(* IEC 61131-3 sources: PortalRobot/Portal_robot/Device/application/FB/FB_MULTI_TYPE, 3 files *)

(* ---- FB_MULTI_TYPE_CONFIG_MANAGER.st ---- *)
FUNCTION_BLOCK FB_MULTI_TYPE_CONFIG_MANAGER
VAR_INPUT
	xTestInitialize  : BOOL; // Атомарная загрузка конфигурации из тестового буфера
	stTestScenario   : ST_TEST_SCENARIO_BUFFER;
	Command          : ST_MULTI_TYPE_COMMAND; // Запросы конфигурации от HMI
	xCellRunning     : BOOL; // Автоматический цикл выполняется
	xMotionBusy      : BOOL; // Оси ещё движутся
	stRobotStatus    : ST_ROBOT_STATUS; // Состояние робота
	astMagazineStatus : ARRAY [1..GVL_CELL_SETTINGS.MagazineCount] OF ST_MAGAZINE_STATUS; // Оба магазина
	astMachineStatus : ARRAY [1..3] OF ST_MACHINE_PUBLIC; // Состояния станков
	uiRows           : UINT; // Строки активной матрицы
	uiColumns        : UINT; // Столбцы активной матрицы
END_VAR
VAR_OUTPUT
	Config : ST_MULTI_TYPE_CONFIG; // Фактически принятая конфигурация
	Status : ST_MULTI_TYPE_CONFIG_STATUS; // Разрешения и диагностика
END_VAR
VAR
	xInitialized        : BOOL; // Начальные безопасные значения заданы
	xAllMachinesSafe    : BOOL; // Станки не обслуживаются и не обрабатывают
	xAllMachinesDisabled: BOOL; // Все станки выключены
	xAllMagazinesEditable : BOOL; // Оба магазина выключены и не заняты
	xAllTypesHaveMachines : BOOL; // Каждый тип назначен хотя бы одному станку
	uiMachine           : UINT; // Индекс станка
	uiMagazine          : UINT; // Индекс магазина
	uiSlot              : UINT; // Индекс слота
	uiType              : UINT; // Индекс типа
	auiMachineCount     : ARRAY [1..3] OF UINT; // Количество станков каждого типа
	auiSlotCount        : ARRAY [1..3] OF UINT; // Количество слотов каждого типа
	rtSetTypeCount      : R_TRIG; // Фронт изменения количества типов
	rtSetMachineType    : R_TRIG; // Фронт назначения типа станку
	rtSetSlotType       : R_TRIG; // Фронт назначения типа слоту
	rtAutoDistribute    : R_TRIG; // Фронт автоматического распределения
END_VAR
VAR CONSTANT
	FIRST_MACHINE : UINT := UINT#1;
	LAST_MACHINE  : UINT := UINT#3;
	FIRST_TYPE    : UINT := UINT#1;
	LAST_TYPE     : UINT := UINT#3;
	WRN_TYPE_COUNT_NOT_ALLOWED : UINT := UINT#23;
	WRN_MACHINE_TYPE_REJECTED  : UINT := UINT#24;
	WRN_SLOT_TYPE_REJECTED     : UINT := UINT#25;
	WRN_DISTRIBUTION_REJECTED  : UINT := UINT#26;
END_VAR

// --- BEGIN IMPLEMENTATION ---

IF (uiRows > UINT#0)
AND (uiColumns > UINT#0)
AND ((uiRows * uiColumns) <= SINT_TO_UINT(GVL_CELL_SETTINGS.NumberDetail)) THEN
	Status.uiActiveSlotCount := uiRows * uiColumns;
ELSE
	Status.uiActiveSlotCount := UINT#0;
END_IF;

IF NOT xInitialized THEN
	Config.uiTypeCount := UINT#1;
	FOR uiMachine := FIRST_MACHINE TO LAST_MACHINE DO
		Config.auiMachineType[uiMachine] := UINT#1;
	END_FOR;
	FOR uiSlot := UINT#1 TO SINT_TO_UINT(GVL_CELL_SETTINGS.NumberDetail) DO
		IF uiSlot <= Status.uiActiveSlotCount THEN
			Config.auiSlotType[uiSlot] := UINT#1;
		ELSE
			Config.auiSlotType[uiSlot] := UINT#0;
		END_IF;
	END_FOR;
	xInitialized := TRUE;
END_IF;

xAllMachinesSafe := TRUE;
xAllMachinesDisabled := TRUE;
FOR uiMachine := FIRST_MACHINE TO LAST_MACHINE DO
	IF astMachineStatus[uiMachine].xBusy
	OR astMachineStatus[uiMachine].xProcessing THEN
		xAllMachinesSafe := FALSE;
	END_IF;
	IF astMachineStatus[uiMachine].xEnabled
	OR astMachineStatus[uiMachine].xDisablePending THEN
		xAllMachinesDisabled := FALSE;
	END_IF;
END_FOR;

xAllMagazinesEditable := TRUE;
FOR uiMagazine := UINT#1 TO INT_TO_UINT(GVL_CELL_SETTINGS.MagazineCount) DO
	IF astMagazineStatus[uiMagazine].xEnabled
	OR astMagazineStatus[uiMagazine].xBusy
	OR astMagazineStatus[uiMagazine].xDisablePending THEN
		xAllMagazinesEditable := FALSE;
	END_IF;
END_FOR;

Status.xMagazineConfigAllowed := NOT xCellRunning
	AND NOT xMotionBusy
	AND NOT stRobotStatus.xBusy
	AND NOT stRobotStatus.xBlankAvailable
	AND NOT stRobotStatus.xDetailAvailable
	AND xAllMagazinesEditable
	AND xAllMachinesSafe;
Status.xTypeCountAllowed := Status.xMagazineConfigAllowed
	AND xAllMachinesDisabled;

FOR uiMachine := FIRST_MACHINE TO LAST_MACHINE DO
	Status.axMachineTypeAllowed[uiMachine] := NOT xCellRunning
		AND NOT xMotionBusy
		AND NOT stRobotStatus.xBusy
		AND NOT stRobotStatus.xBlankAvailable
		AND NOT stRobotStatus.xDetailAvailable
		AND xAllMagazinesEditable
		AND NOT astMachineStatus[uiMachine].xEnabled
		AND NOT astMachineStatus[uiMachine].xDisablePending
		AND NOT astMachineStatus[uiMachine].xBusy
		AND NOT astMachineStatus[uiMachine].xProcessing;
END_FOR;

rtSetTypeCount(CLK := Command.xSetTypeCount);
rtSetMachineType(CLK := Command.xSetMachineType);
rtSetSlotType(CLK := Command.xSetSlotType);
rtAutoDistribute(CLK := Command.xAutoDistribute);

IF rtSetTypeCount.Q THEN
	IF NOT Status.xTypeCountAllowed
	OR (Command.uiRequestedTypeCount < FIRST_TYPE)
	OR (Command.uiRequestedTypeCount > LAST_TYPE) THEN
		RaiseWarning(uiCode := WRN_TYPE_COUNT_NOT_ALLOWED);
	ELSE
		Config.uiTypeCount := Command.uiRequestedTypeCount;
		CASE Config.uiTypeCount OF
			UINT#1:
				Config.auiMachineType[1] := UINT#1;
				Config.auiMachineType[2] := UINT#1;
				Config.auiMachineType[3] := UINT#1;
			UINT#2:
				Config.auiMachineType[1] := UINT#1;
				Config.auiMachineType[2] := UINT#1;
				Config.auiMachineType[3] := UINT#2;
			UINT#3:
				Config.auiMachineType[1] := UINT#1;
				Config.auiMachineType[2] := UINT#2;
				Config.auiMachineType[3] := UINT#3;
		END_CASE;
		ApplyDistribution();
	END_IF;
END_IF;

IF rtSetMachineType.Q THEN
	IF (Command.uiRequestedMachine < FIRST_MACHINE)
	OR (Command.uiRequestedMachine > LAST_MACHINE) THEN
		RaiseWarning(uiCode := WRN_MACHINE_TYPE_REJECTED);
	ELSE
		IF (Command.uiRequestedMachineType < FIRST_TYPE)
		OR (Command.uiRequestedMachineType > Config.uiTypeCount)
		OR NOT Status.axMachineTypeAllowed[Command.uiRequestedMachine] THEN
			RaiseWarning(uiCode := WRN_MACHINE_TYPE_REJECTED);
		ELSE
			Config.auiMachineType[Command.uiRequestedMachine] := Command.uiRequestedMachineType;
		END_IF;
	END_IF;
END_IF;

IF rtSetSlotType.Q THEN
	IF NOT Status.xMagazineConfigAllowed
	OR (Command.uiRequestedSlot < UINT#1)
	OR (Command.uiRequestedSlot > Status.uiActiveSlotCount)
	OR (Command.uiRequestedSlotType < FIRST_TYPE)
	OR (Command.uiRequestedSlotType > Config.uiTypeCount) THEN
		RaiseWarning(uiCode := WRN_SLOT_TYPE_REJECTED);
	ELSE
		Config.auiSlotType[Command.uiRequestedSlot] := Command.uiRequestedSlotType;
	END_IF;
END_IF;

IF rtAutoDistribute.Q THEN
	xAllTypesHaveMachines := TRUE;
	FOR uiType := FIRST_TYPE TO LAST_TYPE DO
		auiMachineCount[uiType] := UINT#0;
	END_FOR;
	FOR uiMachine := FIRST_MACHINE TO LAST_MACHINE DO
		IF (Config.auiMachineType[uiMachine] >= FIRST_TYPE)
		AND (Config.auiMachineType[uiMachine] <= Config.uiTypeCount) THEN
			auiMachineCount[Config.auiMachineType[uiMachine]] :=
				auiMachineCount[Config.auiMachineType[uiMachine]] + UINT#1;
		END_IF;
	END_FOR;
	FOR uiType := FIRST_TYPE TO Config.uiTypeCount DO
		IF auiMachineCount[uiType] = UINT#0 THEN
			xAllTypesHaveMachines := FALSE;
		END_IF;
	END_FOR;

	IF NOT Status.xMagazineConfigAllowed
	OR NOT xAllTypesHaveMachines THEN
		RaiseWarning(uiCode := WRN_DISTRIBUTION_REJECTED);
	ELSE
		ApplyDistribution();
	END_IF;
END_IF;

// Тестовый сценарий проходит общую PLC-валидацию до этого вызова. Запись
// выполняет владелец Config, поэтому значения не теряются на выходной привязке FB.
IF xTestInitialize THEN
	Config.uiTypeCount := stTestScenario.uiTypeCount;
	FOR uiMachine := FIRST_MACHINE TO LAST_MACHINE DO
		Config.auiMachineType[uiMachine] := stTestScenario.auiMachineType[uiMachine];
	END_FOR;
	FOR uiSlot := UINT#1 TO SINT_TO_UINT(GVL_CELL_SETTINGS.NumberDetail) DO
		Config.auiSlotType[uiSlot] := stTestScenario.auiSlotType[uiSlot];
	END_FOR;
END_IF;

FOR uiType := FIRST_TYPE TO LAST_TYPE DO
	auiMachineCount[uiType] := UINT#0;
	auiSlotCount[uiType] := UINT#0;
END_FOR;

Status.xConfigurationValid := (Config.uiTypeCount >= FIRST_TYPE)
	AND (Config.uiTypeCount <= LAST_TYPE)
	AND (Status.uiActiveSlotCount > UINT#0);

FOR uiMachine := FIRST_MACHINE TO LAST_MACHINE DO
	IF (Config.auiMachineType[uiMachine] < FIRST_TYPE)
	OR (Config.auiMachineType[uiMachine] > Config.uiTypeCount) THEN
		Status.xConfigurationValid := FALSE;
	ELSE
		auiMachineCount[Config.auiMachineType[uiMachine]] :=
			auiMachineCount[Config.auiMachineType[uiMachine]] + UINT#1;
	END_IF;
END_FOR;

FOR uiSlot := UINT#1 TO Status.uiActiveSlotCount DO
	IF (Config.auiSlotType[uiSlot] < FIRST_TYPE)
	OR (Config.auiSlotType[uiSlot] > Config.uiTypeCount) THEN
		Status.xConfigurationValid := FALSE;
	ELSE
		auiSlotCount[Config.auiSlotType[uiSlot]] :=
			auiSlotCount[Config.auiSlotType[uiSlot]] + UINT#1;
	END_IF;
END_FOR;

FOR uiType := FIRST_TYPE TO Config.uiTypeCount DO
	IF (auiMachineCount[uiType] = UINT#0)
	OR (auiSlotCount[uiType] = UINT#0) THEN
		Status.xConfigurationValid := FALSE;
	END_IF;
END_FOR;

(* ---- FB_MULTI_TYPE_CONFIG_MANAGER.ApplyDistribution.st ---- *)
METHOD PRIVATE ApplyDistribution
VAR
	uiMachine       : UINT; // Индекс станка
	uiType          : UINT; // Индекс типа
	uiSlot          : UINT; // Индекс слота
	uiAssigned      : UINT; // Число уже назначенных слотов
	uiRemaining     : UINT; // Остаток после целочисленного деления
	uiBestType      : UINT; // Тип с наибольшей дробной частью
	uiBestRemainder : UINT; // Наибольшая дробная часть
	auiMachineShare : ARRAY [1..3] OF UINT; // Число станков типа
	auiQuota        : ARRAY [1..3] OF UINT; // Число слотов типа
	auiRemainder    : ARRAY [1..3] OF UINT; // Остаток квоты
	axExtraAssigned : ARRAY [1..3] OF BOOL; // Дополнительный слот уже выдан типу
END_VAR

// --- BEGIN IMPLEMENTATION ---

FOR uiType := UINT#1 TO UINT#3 DO
	auiMachineShare[uiType] := UINT#0;
	auiQuota[uiType] := UINT#0;
	auiRemainder[uiType] := UINT#0;
	axExtraAssigned[uiType] := FALSE;
END_FOR;

FOR uiMachine := UINT#1 TO UINT#3 DO
	IF (Config.auiMachineType[uiMachine] >= UINT#1)
	AND (Config.auiMachineType[uiMachine] <= Config.uiTypeCount) THEN
		auiMachineShare[Config.auiMachineType[uiMachine]] :=
			auiMachineShare[Config.auiMachineType[uiMachine]] + UINT#1;
	END_IF;
END_FOR;

uiAssigned := UINT#0;
FOR uiType := UINT#1 TO Config.uiTypeCount DO
	auiQuota[uiType] := (Status.uiActiveSlotCount * auiMachineShare[uiType]) / UINT#3;
	auiRemainder[uiType] := (Status.uiActiveSlotCount * auiMachineShare[uiType]) MOD UINT#3;
	uiAssigned := uiAssigned + auiQuota[uiType];
END_FOR;

uiRemaining := Status.uiActiveSlotCount - uiAssigned;
WHILE uiRemaining > UINT#0 DO
	uiBestType := UINT#0;
	uiBestRemainder := UINT#0;
	FOR uiType := UINT#1 TO Config.uiTypeCount DO
		IF NOT axExtraAssigned[uiType]
		AND ((uiBestType = UINT#0) OR (auiRemainder[uiType] > uiBestRemainder)) THEN
			uiBestType := uiType;
			uiBestRemainder := auiRemainder[uiType];
		END_IF;
	END_FOR;
	IF uiBestType = UINT#0 THEN
		uiBestType := UINT#1;
	END_IF;
	auiQuota[uiBestType] := auiQuota[uiBestType] + UINT#1;
	axExtraAssigned[uiBestType] := TRUE;
	uiRemaining := uiRemaining - UINT#1;
END_WHILE;

uiSlot := UINT#1;
FOR uiType := UINT#1 TO Config.uiTypeCount DO
	uiAssigned := UINT#0;
	WHILE (uiAssigned < auiQuota[uiType])
	AND (uiSlot <= Status.uiActiveSlotCount) DO
		Config.auiSlotType[uiSlot] := uiType;
		uiAssigned := uiAssigned + UINT#1;
		uiSlot := uiSlot + UINT#1;
	END_WHILE;
END_FOR;

FOR uiSlot := Status.uiActiveSlotCount + UINT#1 TO SINT_TO_UINT(GVL_CELL_SETTINGS.NumberDetail) DO
	Config.auiSlotType[uiSlot] := UINT#0;
END_FOR;

(* ---- FB_MULTI_TYPE_CONFIG_MANAGER.RaiseWarning.st ---- *)
METHOD PRIVATE RaiseWarning
VAR_INPUT
	uiCode : UINT; // Код отклонённой команды конфигурации
END_VAR

// --- BEGIN IMPLEMENTATION ---

Status.stWarning.uiCode := uiCode;
Status.stWarning.udiSequence := Status.stWarning.udiSequence + UDINT#1;
IF Status.stWarning.udiSequence = UDINT#0 THEN
	Status.stWarning.udiSequence := UDINT#1;
END_IF;
